# EPICS IOC start-up script: iocBoot/iocxxx/examples/detectors/ADProsilica.iocsh
#- INSTANCE  - Used for Camera Port Name and detector pv name
#- ID        - Camera ID or IP address
#- XSIZE     - Image Width
#- YSIZE     - Image Height
#- TYPE      - Image Datatype, default: Int8
#- COLORS    - Number of colors, default: 1

epicsEnvSet("EPICS_DB_INCLUDE_PATH", "$(EPICS_DB_INCLUDE_PATH):$(ADCORE)/db:$(ADPROSILICA)/db")

#- prosilicaConfig(portName,    # The name of the asyn port to be created
#-                 cameraId,    # Unique ID, IP address, or IP name of the camera
#-                 maxBuffers,  # Maximum number of NDArray buffers driver can allocate. 0=unlimited
#-                 maxMemory,   # Maximum memory bytes driver can allocate. 0=unlimited
#-                 priority,    # EPICS thread priority for asyn port driver 0=default
#-                 stackSize,   # EPICS thread stack size for asyn port driver 0=default
#-                 maxPvAPIFrames) # Number of frames to allocate in PvAPI driver. Default=2.
#- The simplest way to determine the uniqueId of a camera is to run the Prosilica GigEViewer application,
#- select the camera, and press the "i" icon on the bottom of the main window to show the camera information for this camera.
#- The Unique ID will be displayed on the first line in the information window.

prosilicaConfig("$(INSTANCE)", "$(ID)", 50, 0)
dbLoadRecords("$(ADPROSILICA)/db/prosilica.template","P=$(PREFIX),R=$(INSTANCE):,PORT=$(INSTANCE),ADDR=0,TIMEOUT=1")

# Create a standard arrays plugin
NDStdArraysConfigure("Image1", 3, 0, "$(INSTANCE)", 0, 2000000)

# Need to determine certain values from input parameters
iocshRun('epicsEnvSet("__FTVL", "$($(TYPE=Int8)_VAL)")', "Int8_VAL=UCHAR, UInt8_VAL=UCHAR, Int16_VAL=SHORT, UInt16_VAL=SHORT, Int32_VAL=LONG, UInt32_VAL=LONG, Float32_VAL=DOUBLE, Float64_VAL=DOUBLE")
iocshRun('epicsEnvSet("__TYPE", "$($(TYPE=Int8)_VAL)")', "Int8_VAL=Int8, UInt8_VAL=Int8, Int16_VAL=Int16, UInt16_VAL=Int16, Int32_VAL=Int32, UInt32_VAL=Int32, Float32_VAL=Float32, Float64_VAL=Float64")
iocshRun('epicsEnvSet("__BYTES", "$($(TYPE=Int8)_VAL)")', "Int8_VAL=1, UInt8_VAL=1, Int16_VAL=2, UInt16_VAL=2, Int32_VAL=4, UInt32_VAL=4, Float32_VAL=4, Float64_VAL=8")
luaCmd("epicsEnvSet('__SIZE', tostring((COLORS*XSIZE*YSIZE)|0))", "COLORS=$(COLORS=1), XSIZE=$(XSIZE), YSIZE=$(YSIZE)")
luaCmd("epicsEnvSet('EPICS_CA_MAX_ARRAY_BYTES', tostring(math.ceil(1.1 * SIZE * BYTES)))", "SIZE=$(__SIZE), BYTES=$(__BYTES)")

dbLoadRecords("$(ADCORE)/ADApp/Db/NDStdArrays.template", "P=$(PREFIX),R=image1:,PORT=Image1,ADDR=0,TIMEOUT=1,NDARRAY_PORT=$(INSTANCE),TYPE=$(__TYPE),FTVL=$(__FTVL),NELEMENTS=$(__SIZE)")

epicsEnvUnset("__FTVL")
epicsEnvUnset("__TYPE")
epicsEnvUnset("__BYTES")
epicsEnvUnset("__SIZE")

iocshLoad("$(ADCORE)/iocBoot/commonPlugins.cmd", "PREFIX=$(PREFIX), PORT=$(INSTANCE), QSIZE=20, XSIZE=$(XSIZE), YSIZE=$(YSIZE), NCHANS=1024, CBUFFS=20, MAX_THREADS=5")

set_requestfile_path("$(ADPROSILICA)/db")
